//EL5021 | 1-channel Sin/Cos encoder
FUNCTION_BLOCK EL5021

VAR_INPUT
	En: BOOL;
	iTerminal_ID : INT;
	ErrorSystem : POINTER TO ST_ErrorSystem;
END_VAR

VAR_OUTPUT
	EnO: BOOL;
	Counter_Value : UDINT;
	Latch_Value : UDINT;
	bError: BOOL;
END_VAR

VAR
	udiCounter_Value AT %I* : UDINT;
	udiLatch_Value AT %I* : UDINT;
	WcState_WcState AT %I*: BOOL;
	InfoData_State AT %I*: UINT;
	
	//FB-s
	fbTerminalError : FB_TerminalError;
END_VAR

(*
* TODO:
* Channel Status words, control words
*)

EnO:=En;

//Error FB instance
fbTerminalError(
	En := TRUE,
	iTerminal_ID := iTerminal_ID,
	bWcState := WcState_WcState,
	uiInfoData_State := InfoData_State,
	pErrorSystem := ErrorSystem,
	bError => bError,
);

IF EN THEN
	IF NOT bError THEN
		Counter_Value := udiCounter_Value;
		Latch_Value := udiLatch_Value;
	ELSE
		Counter_Value := 0;
		Latch_Value := 0;
	END_IF
END_IF

END_FUNCTION_BLOCK

(* stored: Version 1.1.0.1, ProductVersion 3.1.4022.10
   POU EL5021: Id {7f517c2d-3257-42d3-9c58-98a243359439}, SpecialFunc None *)
